FUNCTION_BLOCK FB_Cylinder_1 IMPLEMENTS ITF_Cylinder
VAR
	_atHomePos AT %I* : BOOL; // Link With Home Position Sensor
	_atWorkPos AT %I* : BOOL; // Link With Work Position Sensor
	toHomePos AT %Q* : BOOL;
	toWorkPos AT %Q* : BOOL;
	
	{attribute 'hide'}
	_simulate : BOOL := TRUE;
	simTimer : TON := ( PT := CYLINDER_MOVE_TIME );
END_VAR
VAR CONSTANT
	CYLINDER_MOVE_TIME : TIME := T#1S;
END_VAR

PROPERTY AtHome : bool
GET
AtHome := _atHomePos OR_ELSE simTimer.Q;
simTimer( IN := _simulate AND_THEN toHomePos );
END_GET
END_PROPERTY

PROPERTY AtWork : bool
GET
AtWork := _atWorkPos OR_ELSE simTimer.Q;
simTimer( IN := _simulate AND_THEN toWorkPos );
END_GET
END_PROPERTY

METHOD MoveToHome
toHomePos := TRUE;
toWorkPos := FALSE; 
simTimer( IN := FALSE );
END_METHOD

/// Move To Work Position
METHOD MoveToWork
VAR_INPUT
END_VAR
toWorkPos := TRUE; 
toHomePos := FALSE;
simTimer( IN := FALSE );
END_METHOD

PROPERTY MovingToHomePosition : BOOL
GET
MovingToHomePosition := toHomePos AND NOT AtHome;
END_GET
END_PROPERTY

PROPERTY MovingToWorkPosition : BOOL
GET
MovingToWorkPosition := toWorkPos AND NOT AtWork;
END_GET
END_PROPERTY

METHOD PROTECTED SetSimulationMode : BOOL
VAR_INPUT
	Active : BOOL; 
END_VAR
IF (MovingToHomePosition OR MovingToWorkPosition) THEN
	RETURN; // Cannot set simulation while moving.
END_IF

_simulate := Active;
SetSimulationMode := TRUE;
END_METHOD

PROPERTY PUBLIC SimulationActive : BOOL
GET
SimulationActive := _simulate;
END_GET
END_PROPERTY

END_FUNCTION_BLOCK

(* stored: Version 1.1.0.1, ProductVersion 3.1.4024.5
   POU FB_Cylinder_1: Id {4a4d6dd2-5490-43cc-b30a-511aab936e58}, SpecialFunc None
   Folder Methods: Id {421b5337-e995-40fb-aba2-4176c9bf04ca}
   Folder Props: Id {30b8d09f-d264-487c-adac-f704f2f9b675}
   Property AtHome: Id {47da66d8-5d0c-4067-81ec-658d24dc9a7f}
   Get Get: Id {572301e4-3e8a-42cb-9d02-21eef0dea0d1}
   Property AtWork: Id {1f06914f-45b0-42d7-8877-978e867270bb}
   Get Get: Id {ea38930e-f705-4e17-8825-cccebd6aa905}
   Method MoveToHome: Id {371d9fc7-9b6c-4c93-8896-f96284459f17}
   Method MoveToWork: Id {5b531c35-d6d5-4d36-b459-1b66b6844bbe}
   Property MovingToHomePosition: Id {d85f6d6d-1fcd-44a7-a8bb-79beeaebde2c}
   Get Get: Id {fc085a47-c687-46ee-a1c2-ede8b5fd304b}
   Property MovingToWorkPosition: Id {9380a718-018b-480d-9b6f-c32849365348}
   Get Get: Id {87254797-56af-474f-825b-b4807b588849}
   Method SetSimulationMode: Id {e6a68196-9278-4167-a2c5-fa30e330b259}
   Property SimulationActive: Id {ae8171c4-c362-401e-93f2-9371f6bd9dbe}
   Get Get: Id {a3306cc1-987a-4ac4-b09f-681bc64096dd} *)
